TYPE CAN_MSG :
STRUCT
	ID   : UDINT; // Unsigned 32-bit
	DLC  : BYTE;  // Unsigned 8-bit
	DATA : ARRAY[0..7] OF BYTE;
END_STRUCT
END_TYPE

(* stored: Version 1.1.0.1
   DUT CAN_MSG: Id {9211ddd6-2c71-42b3-b63f-ea004e11d2ed} *)
